// TIA Portal V21 export
VAR_GLOBAL   // PLC tag table "ClusterReciveDigitali"
END_VAR
VAR_GLOBAL CONSTANT   // user constants
   K_SegnaleDaCluster_Ready : Int := 1;
   K_SegnaleDaCluster_Marcia : Int := 2;
END_VAR
